{attribute 'qualified_only'}
{attribute 'strict'}
TYPE LaserPlace_e :
(
    NearTrack := 0,
    NearDoor := 1
);
END_TYPE

(* stored: Version 1.1.0.1, ProductVersion 3.1.4024.6
   DUT LaserPlace_e: Id {7129bb50-ba8a-4532-a2ab-58af0193d35c} *)
